PROGRAM PRG_TEST
VAR
	FB_System_Test : FB_System_Test;
	FB_Clamp01_Test : FB_Clamp01_Test;
	FB_Compare_Test : FB_Compare_Test;
	FB_Norm_Test : FB_Norm_Test;
	FB_Scale_Test : FB_Scale_Test;
	FB_Sign_Test : FB_Sign_Test;
	FB_InverBytesOrder_Test : FB_InverBytesOrder_Test;
	FB_GetByte_Test : FB_GetByte_Test;
	FB_Swap_Test : FB_Swap_Test; 
	FB_MEMCPY_Test : FB_MEMCPY_Test;
	FB_Heater_Test : FB_Heater_Test;
	FB_MoveVelocity_Test : FB_MoveVelocity_Test;
	FB_MoveAbsolute_Test : FB_MoveAbsolute_Test; 
	FB_DriveControl_Test : FB_DriveControl_Test;
	FB_Button_Test : FB_Button_Test;
	FB_Switch_Test : FB_Switch_Test;
	FB_Lock_Test : FB_Lock_Test;
	FB_Panel_Test : FB_Panel_Test;
	FB_Cylinder_Test : FB_Cylinder_Test;
	FB_Device_Test : FB_Device_Test;
	FB_DeviceByte_Test : FB_DeviceByte_Test;
	FB_DeviceWord_Test : FB_DeviceWord_Test;
	FB_DeviceDWord_Test : FB_DeviceDWord_Test;
	FB_DeviceLWord_Test : FB_DeviceLWord_Test;
	FB_DeviceReal_Test : FB_DeviceReal_Test;
	FB_Drive_Test : FB_Drive_Test;
	FB_Lamp_Test : FB_Lamp_Test;
	FB_Reader_Test : FB_Reader_Test;
	FB_SensorAnalog_Test : FB_SensorAnalog_Test;
	FB_SensorBinary_Test : FB_SensorBinary_Test;
	FB_Robot_Test : FB_Robot_Test;
	FB_DS402FSM_Test : FB_DS402FSM_Test;
	FB_DS402_Test : FB_DS402_Test;
	FB_Euchner_MGB_Test : FB_Euchner_MGB_Test;
	FB_Euchner_STP_Test : FB_Euchner_STP_Test;
	FB_SimMovitracLTEB_Test : FB_SimMovitracLTEB_Test;
	FB_Starter_Test : FB_Starter_Test;
	FB_SimMovidriveFSM_Test : FB_SimMovidriveFSM_Test;
	FB_SimMovitrac_Test : FB_SimMovitrac_Test;
	FB_SimMovitracB_Test : FB_SimMovitracB_Test;
	FB_AdsMessageHandler_Test : FB_AdsMessageHandler_Test;
	FB_RecordData_Test : FB_RecordData_Test;
	FB_SimMovidrivePDO12_Test : FB_SimMovidrivePDO12_Test;
	FB_Encoder_Test : FB_Encoder_Test;		
END_VAR

TcUnit.RUN();

END_PROGRAM

(* stored: Version 1.1.0.1, ProductVersion 3.1.4024.12
   POU PRG_TEST: Id {3e1b042c-faae-06db-38f4-585c236d1642}, SpecialFunc None *)
